{attribute 'GeneratedUsingTerminal: AX8108-0100-0101-0101'}
{attribute addProperty BoxType "AX8108-0100-0101-0101"}
{attribute addProperty Id "AdsAddrAT %I*AMSADDR8DcOutputShiftAT %I*DINT4DcInputShiftAT %I*DINT4AoeNetIdAT %I*AMSNETID6Chn0AT %I*USINT1StateAT %I*UINT2"}
{attribute addProperty CRC "898259407"}
{attribute addProperty Size "25"}
TYPE InfoData_358A59CF EXTENDS InputBase_8311D824 :
STRUCT
	{attribute addProperty Name "AdsAddr"}
	AdsAddr AT %I* : AMSADDR;
	{attribute addProperty Name "DcOutputShift"}
	DcOutputShift AT %I* : DINT;
	{attribute addProperty Name "DcInputShift"}
	DcInputShift AT %I* : DINT;
	{attribute addProperty Name "AoeNetId"}
	AoeNetId AT %I* : AMSNETID;
	{attribute addProperty Name "Chn0"}
	Chn0 AT %I* : USINT;
	{attribute addProperty Name "State"}
	State AT %I* : UINT;
END_STRUCT
END_TYPE

(* stored: Version 1.2.0.0, ProductVersion 3.1.4024.9
   DUT InfoData_358A59CF: Id {5a7a4909-c513-4cdd-a476-fb853d275f5d} *)
